// TwinCAT 3 PLC project PIDControllerTests
// ProgramVersion: 3.1.4026.22
// libraries:
//   Tc2_Standard, * (Beckhoff Automation GmbH)
//   Tc2_System, * (Beckhoff Automation GmbH)
//   TcUnit, * (www.tcunit.org)
//   B5PIDController_Plc,newest,Tc3 Project
// project tree:
//   / PlcTask.TcTTO
//   POUs/ FB_PIDControllerConsumer.TcPOU, MAIN.TcPOU
// (motion and I/O tree: see PLC project b5pidcontroller_plc)

CONFIGURATION PIDControllerTests
    RESOURCE PLC ON TwinCAT3
        TASK PlcTask(INTERVAL := T#10ms, PRIORITY := 21);
        PROGRAM MAIN WITH PlcTask : MAIN;
    END_RESOURCE
END_CONFIGURATION

// ---- POUs/MAIN.TcPOU
PROGRAM MAIN
VAR
END_VAR

END_PROGRAM

// ---- POUs/FB_PIDControllerConsumer.TcPOU
FUNCTION_BLOCK FB_PIDControllerConsumer
VAR
    controller : B5PIDController_Plc.FB_PIDController;
    output : REAL;
END_VAR

controller(fError := 2.5);
output := controller.Step();

END_FUNCTION_BLOCK
